PROGRAM AlarmInit
VAR
END_VAR

//Stepper Motors Alarms
g_aAlarms[StepperHomingFailed].sMessage := '';
g_aAlarms[StepperPositionUnknown].sMessage := 'Low Flow Alarm';
g_aAlarms[StepperMotionTimedOut].sMessage  := 'Door Open Alarm';

//Linear Actuators Alarms
g_aAlarms[LinearActuatorHomingFailed].sMessage  := 'Emergency Stop';
g_aAlarms[LinearActuatorPositionUnknown].sMessage  := 'PLC Battery Fault';
g_aAlarms[LinearActuatorMotionTimedOut].sMessage  := 'PLC Battery Fault';

//Safety Alarms
g_aAlarms[EStopEnabled].sMessage  := 'Emergency Stop Is Enabled';

END_PROGRAM

(* stored: Version 1.1.0.1, ProductVersion 3.1.4024.14
   POU AlarmInit: Id {5de57df6-e3cf-4e7b-aa3b-e5783cfad859}, SpecialFunc None *)
